SUBAPPLICATION SorterLogic (* Subapplication Type *)
  (* Standard: 61499-2 *)
  (* Version 1.0, 2023-02-03, Maximilian Scharf *)
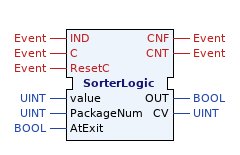
  EVENT_INPUT
    IND;
    C;
    ResetC;
  END_EVENT
  EVENT_OUTPUT
    CNF;
    CNT;
  END_EVENT
  VAR_INPUT
    value : UINT;
    PackageNum : UINT;
    AtExit : BOOL;
  END_VAR
  VAR_OUTPUT
    OUT : BOOL;
    CV : UINT;
  END_VAR
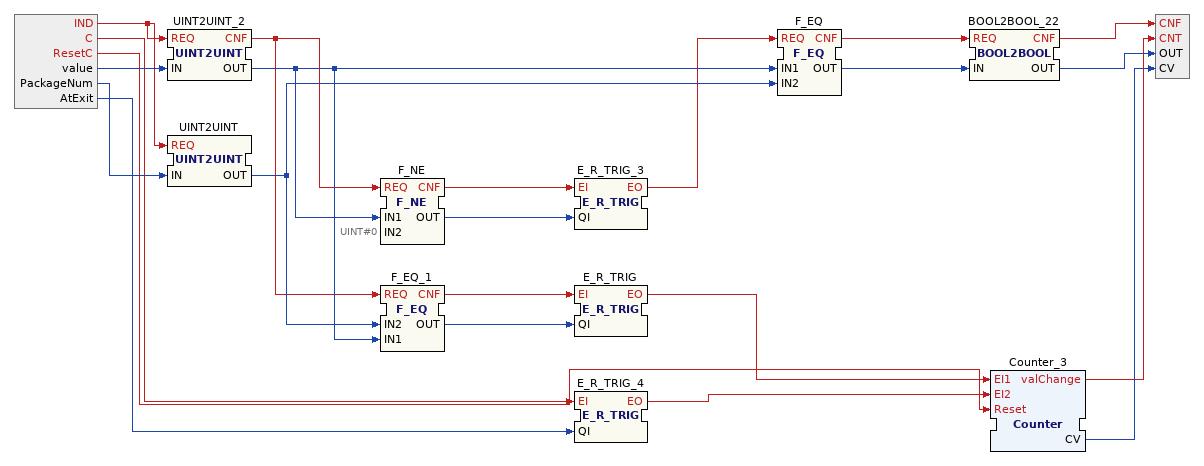
  FBS
    BOOL2BOOL_22 : BOOL2BOOL;
    UINT2UINT_2 : UINT2UINT;
    F_NE : F_NE(IN2 := UINT#0);
    E_R_TRIG_3 : E_R_TRIG;
    F_EQ : F_EQ;
    UINT2UINT : UINT2UINT;
    E_R_TRIG_4 : E_R_TRIG;
    F_EQ_1 : F_EQ;
    E_R_TRIG : E_R_TRIG;
  END_FBS
  SUBAPPS
    Counter_3 : Counter;
  END_SUBAPPS
  EVENT_CONNECTIONS
    F_EQ.CNF TO BOOL2BOOL_22.REQ;
    UINT2UINT_2.CNF TO F_NE.REQ;
    F_NE.CNF TO E_R_TRIG_3.EI;
    E_R_TRIG_3.EO TO F_EQ.REQ;
    BOOL2BOOL_22.CNF TO CNF;
    IND TO UINT2UINT_2.REQ;
    IND TO UINT2UINT.REQ;
    UINT2UINT_2.CNF TO F_EQ_1.REQ;
    E_R_TRIG_4.EO TO Counter_3.EI2;
    F_EQ_1.CNF TO E_R_TRIG.EI;
    E_R_TRIG.EO TO Counter_3.EI1;
    Counter_3.valChange TO CNT;
    C TO E_R_TRIG_4.EI;
    ResetC TO Counter_3.Reset;
  END_CONNECTIONS
  DATA_CONNECTIONS
    F_EQ.OUT TO BOOL2BOOL_22.IN;
    UINT2UINT_2.OUT TO F_NE.IN1;
    UINT2UINT_2.OUT TO F_EQ.IN1;
    F_NE.OUT TO E_R_TRIG_3.QI;
    BOOL2BOOL_22.OUT TO OUT;
    value TO UINT2UINT_2.IN;
    UINT2UINT.OUT TO F_EQ.IN2;
    PackageNum TO UINT2UINT.IN;
    UINT2UINT.OUT TO F_EQ_1.IN2;
    UINT2UINT_2.OUT TO F_EQ_1.IN1;
    F_EQ_1.OUT TO E_R_TRIG.QI;
    AtExit TO E_R_TRIG_4.QI;
    Counter_3.CV TO CV;
  END_CONNECTIONS
END_SUBAPPLICATION
